{attribute 'qualified_only'}
{attribute 'strict'}
{attribute 'to_string'}

TYPE E_EventType :
(
	Alaram := 0,
	Message := 1
);
END_TYPE

(* stored: Version 1.1.0.1, ProductVersion 3.1.4024.16
   DUT E_EventType: Id {c2221df4-0c68-4adc-a193-db714a456f06} *)
